// TIA Portal V20 export
TYPE "typeCmControlNodeCommand"
// stored: Namespace Unit1.Em4
   STRUCT
      sideTapeFixStageAxisX : "LER_typeAxisCommand";
      sideTapeFixStageAxisC : "LER_typeAxisCommand";
      sideTapeAttachmentAxisX { S7_SetPoint := 'True'} : "LER_typeAxisCommand";
      sideTapeAttachmentAxisY { S7_SetPoint := 'True'} : "LER_typeAxisCommand";
      sideTapeLoading { S7_SetPoint := 'True'} : "LER_typeTwoWayActCommand";
      sideTapeLoadingClamp { S7_SetPoint := 'True'} : "LER_typeTwoWayActCommand";
      sideTapeCutter { S7_SetPoint := 'True'} : "LER_typeTwoWayActCommand";
      sideTapeCutterClamp { S7_SetPoint := 'True'} : "LER_typeTwoWayActCommand";
      sideTapeTension { S7_SetPoint := 'True'} : "LER_typeTwoWayActCommand";
      sideTapeAttachmentLeft { S7_SetPoint := 'True'} : "LER_typeTwoWayActCommand";
      sideTapeAttachmentRight { S7_SetPoint := 'True'} : "LER_typeTwoWayActCommand";
      sideTapeAttachmentBtm { S7_SetPoint := 'True'} : "LER_typeTwoWayActCommand";
      sideTapeFixStage { S7_SetPoint := 'True'} : "LER_typeTwoWayActCommand";
      sideTapeAttachmentLeftTopVaccum { S7_SetPoint := 'True'} : "LER_typeTwoWayActCommand";
      sideTapeAttachmentLeftBtmVaccum { S7_SetPoint := 'True'} : "LER_typeTwoWayActCommand";
      sideTapeAttachmentRightTopVaccum { S7_SetPoint := 'True'} : "LER_typeTwoWayActCommand";
      sideTapeAttachmentRightBtmVaccum { S7_SetPoint := 'True'} : "LER_typeTwoWayActCommand";
   END_STRUCT;
END_TYPE
